// TIA Portal V18 export
// export: Created 2025-12-01T12:39:35.6696445Z, ExportSetting None, DisplayName Totally Integrated Automation Portal, DisplayVersion V18 Update 5, DisplayName TIA Portal Openness, DisplayVersion V18 Update 5, DisplayName TIA Portal Teamcenter Gateway, DisplayVersion V18, DisplayName TIA Portal Version Control Interface, DisplayVersion V18, DisplayName STEP 7 Professional, DisplayVersion V18 Update 5, DisplayName STEP 7 Safety, DisplayVersion V18, DisplayName WinCC Professional, DisplayVersion V18 Update 5
VAR_GLOBAL   // PLC tag table "ProcessResult"
END_VAR
VAR_GLOBAL CONSTANT   // user constants
   NO_Part : Int := 0;   // 无产品
   NEW_Part : Int := 100;   // 有料未作业
   Part_boltFinish : Int := 201;   // 顶柱完成
   Part_OK : Int := 400;   // 作业完成，产品OK
   NO_Result : Int := 0;   // 无结果
   OK_Result : Int := 400;   // 结果OK
   NG_Result : Int := 401;   // 结果NG
   Part_SpringFinish : Int := 202;   // 弹簧完成
   Part_TopPostFinish : Int := 203;   // 顶柱完成
   Part_CCDOK : Int := 205;   // 拍照OK
   Part_NG : Int := 401;   // 作业完成，产品NG
   Part_PositionNG : Int := 402;   // 产品姿态NG
   Part_Process : Int := 200;   // 加工中
END_VAR
